Staubli VAL3: PentaclePoint.pgx

public program PentaclePoint(trsf& x_trSource[], trsf& x_trDest[], bool& x_bRes)
  local num l_ni
  local frame l_fFrame
  local num l_Dia
  local num l_nLegth
  local point l_pBuff
  local trsf l_trBuff[3]
  local num l_nNum
begin
  //五角星

  //根据三个trsf建立frame
  call SetFrame(x_trSource,l_fFrame,x_bRes)
  if !x_bRes
    return
  endIf


  //圆弧的直径
  l_nLegth=distance(x_trSource[0],x_trSource[1])

  link(l_pBuff,l_fFrame)
  l_pBuff.trsf={l_nLegth/2,tan(54)*l_nLegth/2,0,0,0,0}
  l_trBuff[0]=position(l_pBuff,world)

  l_pBuff.trsf={l_nLegth/2,tan(36)*l_nLegth/2,0,0,0,0}
  l_trBuff[1]=position(l_pBuff,world)

  l_pBuff.trsf={l_nLegth,0,0,0,0,0}
  l_trBuff[2]=position(l_pBuff,world)

  //根据求的三点建立新的frame
    call SetFrame(l_trBuff,l_fFrame,x_bRes)
  if !x_bRes
    return
  endIf
  l_Dia=distance(l_trBuff[0],l_trBuff[1])
  l_nLegth=distance(l_trBuff[0],l_trBuff[2])


    link(l_pBuff,l_fFrame)
   for l_ni=0 to 9
    l_nNum=sel(l_ni%2==0,l_Dia,l_nLegth)
    l_pBuff.trsf={l_nNum*cos(36*l_ni),sin(36*l_ni)*l_nNum,0,0,0,0}
    x_trDest[l_ni]=position(l_pBuff,world)
  endFor
   x_trDest[10]=x_trDest[0]



end
